// Mitsubishi GX Works2 project: SmartFarmDXnotST   PLC: FX3U/FX3UC

// global labels: Global1
VAR_GLOBAL
  AmbSens1_Humid AT D10 : INT;
  AmbSens1_Temp AT D11 : INT;
  AmbSens2_Humid AT D12 : INT;
  AmbSens2_Temp AT D13 : INT;
  SoilSens1_moist AT D20 : INT;
  SoilSens1_temp AT D21 : INT;
  SoilSens1_cond AT D22 : INT;
  SoilSens1_PH AT D23 : INT;
  SoilSens1_N AT D24 : INT;
  SoilSens1_P AT D25 : INT;
  SoilSens1_K AT D26 : INT;
  TempCon1_minT AT D30 : INT;
  TempCon1_maxT AT D31 : INT;
  TempCon1_Flg AT M10 : BOOL;
  TempCon1_Hs AT D32 : INT;
  TempCon1_Ms AT D33 : INT;
  TempCon1_Ss AT D34 : INT;
  TempCon1_He AT D35 : INT;
  TempCon1_Me AT D36 : INT;
  TempCon1_Se AT D37 : INT;
  TempCon2_minT AT D38 : INT;
  TempCon2_maxT AT D39 : INT;
  TempCon2_Flg AT M20 : BOOL;
  TempCon2_Hs AT D40 : INT;
  TempCon2_Ms AT D41 : INT;
  TempCon2_Ss AT D42 : INT;
  TempCon2_He AT D43 : INT;
  TempCon2_Me AT D44 : INT;
  TempCon2_Se AT D45 : INT;
  HumidCon1_minH AT D46 : INT;
  HumidCon1_maxH AT D47 : INT;
  HumidCon1_Flg AT M30 : BOOL;
  HumidCon1_Hs AT D48 : INT;
  HumidCon1_Ms AT D49 : INT;
  HumidCon1_Ss AT D50 : INT;
  HumidCon1_He AT D51 : INT;
  HumidCon1_Me AT D52 : INT;
  HumidCon1_Se AT D53 : INT;
  HumidCon2_minH AT D54 : INT;
  HumidCon2_maxH AT D55 : INT;
  HumidCon2_Flg AT M40 : BOOL;
  HumidCon2_Hs AT D56 : INT;
  HumidCon2_Ms AT D57 : INT;
  HumidCon2_Ss AT D58 : INT;
  HumidCon2_He AT D59 : INT;
  HumidCon2_Me AT D60 : INT;
  HumidCon2_Se AT D61 : INT;
  TimeCon1_Flg AT M50 : BOOL;
  TimeCon1_Hs AT D62 : INT;
  TimeCon1_Ms AT D63 : INT;
  TimeCon1_Ss AT D64 : INT;
  TimeCon1_He AT D65 : INT;
  TimeCon1_Me AT D66 : INT;
  TimeCon1_Se AT D67 : INT;
  TimeCon2_Flg AT M60 : BOOL;
  TimeCon2_Hs AT D68 : INT;
  TimeCon2_Ms AT D69 : INT;
  TimeCon2_Ss AT D70 : INT;
  TimeCon2_He AT D71 : INT;
  TimeCon2_Me AT D72 : INT;
  TimeCon2_Se AT D73 : INT;
  TimeCon3_Flg AT M70 : BOOL;
  TimeCon3_Hs AT D74 : INT;
  TimeCon3_Ms AT D75 : INT;
  TimeCon3_Ss AT D76 : INT;
  TimeCon3_He AT D77 : INT;
  TimeCon3_Me AT D78 : INT;
  TimeCon3_Se AT D79 : INT;
  TimeCon4_Flg AT M80 : BOOL;
  TimeCon4_Hs AT D80 : INT;
  TimeCon4_Ms AT D81 : INT;
  TimeCon4_Ss AT D82 : INT;
  TimeCon4_He AT D83 : INT;
  TimeCon4_Me AT D84 : INT;
  TimeCon4_Se AT D85 : INT;
  v0_enb AT M100 : BOOL;
  v0_mode_slc AT M101 : BOOL;
  v0_man_OD AT M102 : BOOL;
  v0_Temp1 AT M103 : BOOL;
  v0_Temp2 AT M104 : BOOL;
  v0_Humid1 AT M105 : BOOL;
  v0_Humid2 AT M106 : BOOL;
  v0_Time1 AT M107 : BOOL;
  v0_Time2 AT M108 : BOOL;
  v0_Time3 AT M109 : BOOL;
  v0_Time4 AT M110 : BOOL;
  v0_AMB_config AT M111 : BOOL;
  v0_TIME_config AT M112 : BOOL;
  v0_con_kill_flg AT M113 : BOOL;
  v0_con_pass_flg AT M114 : BOOL;
  v0_Drv_flg AT M115 : BOOL;
  v0_Yman_OD AT M116 : BOOL;
  v0_run_dur AT D100 : INT;
  v0_rest_dur AT D101 : INT;
  v1_enb AT M130 : BOOL;
  v1_mode_slc AT M131 : BOOL;
  v1_man_OD AT M132 : BOOL;
  v1_Temp1 AT M133 : BOOL;
  v1_Temp2 AT M134 : BOOL;
  v1_Humid1 AT M135 : BOOL;
  v1_Humid2 AT M136 : BOOL;
  v1_Time1 AT M137 : BOOL;
  v1_Time2 AT M138 : BOOL;
  v1_Time3 AT M139 : BOOL;
  v1_Time4 AT M140 : BOOL;
  v1_AMB_config AT M141 : BOOL;
  v1_TIME_config AT M142 : BOOL;
  v1_con_kill_flg AT M143 : BOOL;
  v1_con_pass_flg AT M144 : BOOL;
  v1_Drv_flg AT M145 : BOOL;
  v1_Yman_OD AT M146 : BOOL;
  v1_run_dur AT D102 : INT;
  v1_rest_dur AT D103 : INT;
END_VAR

PROGRAM MAIN
VAR
  AmbientSenseRea1 : AmbientSenseRead;
  SoilSenseRead_1 : SoilSenseRead;
  TempCon_1 : TempCon;
  TempCon_2 : TempCon;
  HumidCon_1 : HumidCon;
  HumidCon_2 : HumidCon;
  TimeCon_1 : TimeCon;
  TimeCon_2 : TimeCon;
  TimeCon_3 : TimeCon;
  TimeCon_4 : TimeCon;
  Valve_1 : Valve;
END_VAR
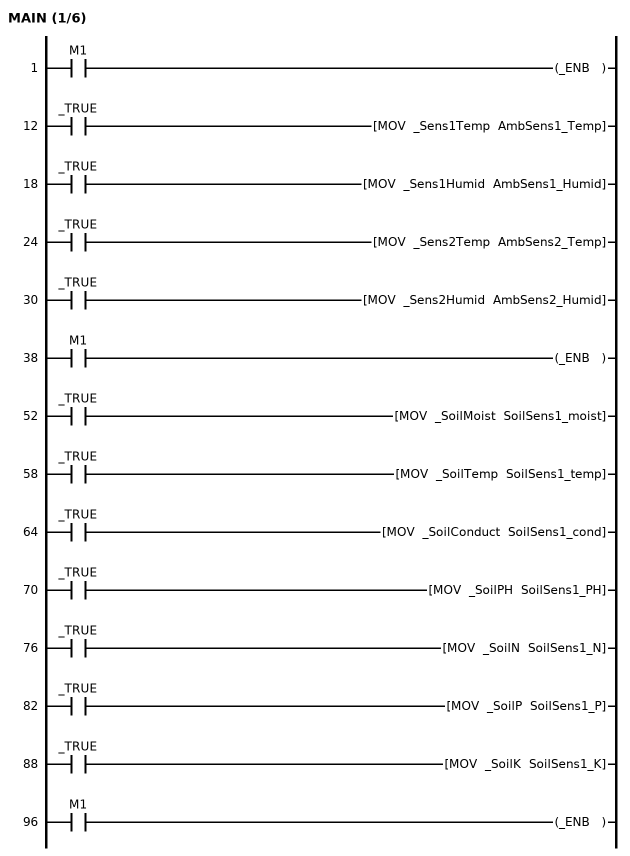
; FB BLK START AmbientSenseRead(AmbientSenseRea1)
1     LD      M1
      OUT     _ENB
; FB START
; FB_NAME AmbientSenseRead
; INSTANCE_NAME AmbientSenseRea1
; FB IN_B:ENB
; FB OUT_Sens1Temp:W
; FB OUT_Sens1Humid:W
; FB OUT_Sens2Temp:W
; FB OUT_Sens2Humid:W
; FB END
12    LD      _TRUE
      MOV     _Sens1Temp AmbSens1_Temp
18    LD      _TRUE
      MOV     _Sens1Humid AmbSens1_Humid
24    LD      _TRUE
      MOV     _Sens2Temp AmbSens2_Temp
30    LD      _TRUE
      MOV     _Sens2Humid AmbSens2_Humid
; FB BLK END
; FB BLK START SoilSenseRead(SoilSenseRead_1)
38    LD      M1
      OUT     _ENB
; FB START
; FB_NAME SoilSenseRead
; INSTANCE_NAME SoilSenseRead_1
; FB IN_B:ENB
; FB OUT_SoilMoist:W
; FB OUT_SoilTemp:W
; FB OUT_SoilConduct:W
; FB OUT_SoilPH:W
; FB OUT_SoilN:W
; FB OUT_SoilP:W
; FB OUT_SoilK:W
; FB END
52    LD      _TRUE
      MOV     _SoilMoist SoilSens1_moist
58    LD      _TRUE
      MOV     _SoilTemp SoilSens1_temp
64    LD      _TRUE
      MOV     _SoilConduct SoilSens1_cond
70    LD      _TRUE
      MOV     _SoilPH SoilSens1_PH
76    LD      _TRUE
      MOV     _SoilN SoilSens1_N
82    LD      _TRUE
      MOV     _SoilP SoilSens1_P
88    LD      _TRUE
      MOV     _SoilK SoilSens1_K
; FB BLK END
; FB BLK START TempCon(TempCon_1)
96    LD      M1
      OUT     _ENB
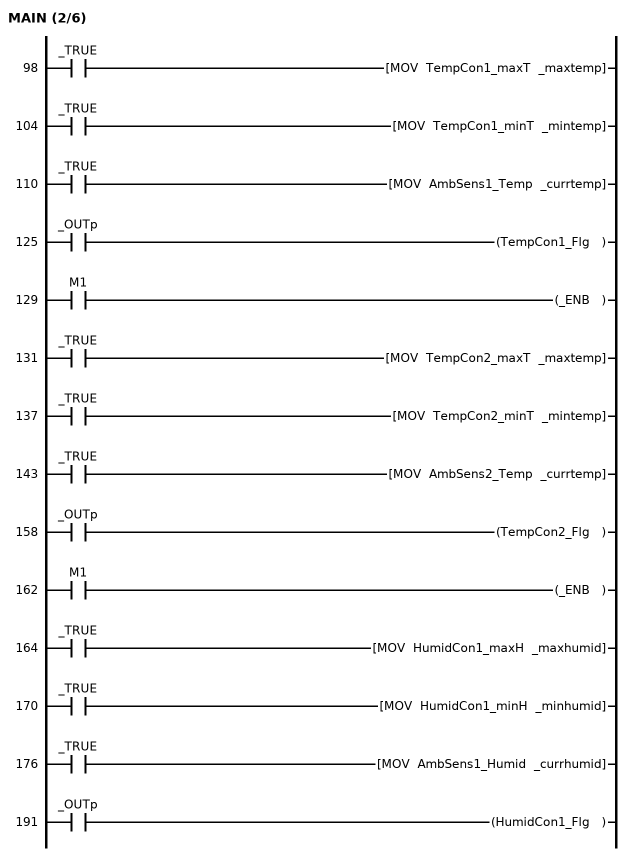
98    LD      _TRUE
      MOV     TempCon1_maxT _maxtemp
104   LD      _TRUE
      MOV     TempCon1_minT _mintemp
110   LD      _TRUE
      MOV     AmbSens1_Temp _currtemp
; FB START
; FB_NAME TempCon
; INSTANCE_NAME TempCon_1
; FB IN_B:ENB
; FB OUT_OUTp:B
; FB IN_W:maxtemp
; FB IN_W:mintemp
; FB IN_W:currtemp
; FB END
125   LD      _OUTp
      OUT     TempCon1_Flg
; FB BLK END
; FB BLK START TempCon(TempCon_2)
129   LD      M1
      OUT     _ENB
131   LD      _TRUE
      MOV     TempCon2_maxT _maxtemp
137   LD      _TRUE
      MOV     TempCon2_minT _mintemp
143   LD      _TRUE
      MOV     AmbSens2_Temp _currtemp
; FB START
; FB_NAME TempCon
; INSTANCE_NAME TempCon_2
; FB IN_B:ENB
; FB OUT_OUTp:B
; FB IN_W:maxtemp
; FB IN_W:mintemp
; FB IN_W:currtemp
; FB END
158   LD      _OUTp
      OUT     TempCon2_Flg
; FB BLK END
; FB BLK START HumidCon(HumidCon_1)
162   LD      M1
      OUT     _ENB
164   LD      _TRUE
      MOV     HumidCon1_maxH _maxhumid
170   LD      _TRUE
      MOV     HumidCon1_minH _minhumid
176   LD      _TRUE
      MOV     AmbSens1_Humid _currhumid
; FB START
; FB_NAME HumidCon
; INSTANCE_NAME HumidCon_1
; FB IN_B:ENB
; FB OUT_OUTp:B
; FB IN_W:maxhumid
; FB IN_W:minhumid
; FB IN_W:currhumid
; FB END
191   LD      _OUTp
      OUT     HumidCon1_Flg
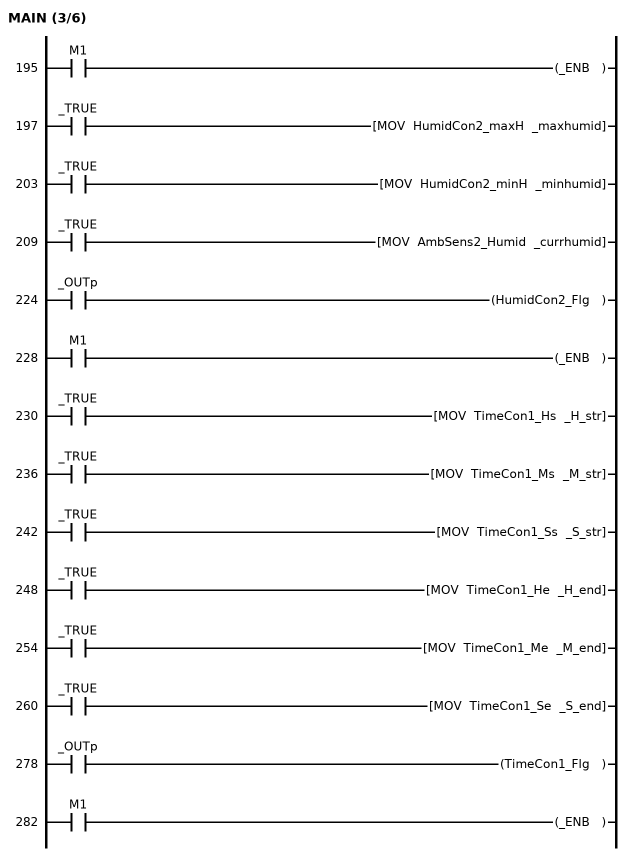
; FB BLK END
; FB BLK START HumidCon(HumidCon_2)
195   LD      M1
      OUT     _ENB
197   LD      _TRUE
      MOV     HumidCon2_maxH _maxhumid
203   LD      _TRUE
      MOV     HumidCon2_minH _minhumid
209   LD      _TRUE
      MOV     AmbSens2_Humid _currhumid
; FB START
; FB_NAME HumidCon
; INSTANCE_NAME HumidCon_2
; FB IN_B:ENB
; FB OUT_OUTp:B
; FB IN_W:maxhumid
; FB IN_W:minhumid
; FB IN_W:currhumid
; FB END
224   LD      _OUTp
      OUT     HumidCon2_Flg
; FB BLK END
; FB BLK START TimeCon(TimeCon_1)
228   LD      M1
      OUT     _ENB
230   LD      _TRUE
      MOV     TimeCon1_Hs _H_str
236   LD      _TRUE
      MOV     TimeCon1_Ms _M_str
242   LD      _TRUE
      MOV     TimeCon1_Ss _S_str
248   LD      _TRUE
      MOV     TimeCon1_He _H_end
254   LD      _TRUE
      MOV     TimeCon1_Me _M_end
260   LD      _TRUE
      MOV     TimeCon1_Se _S_end
; FB START
; FB_NAME TimeCon
; INSTANCE_NAME TimeCon_1
; FB IN_B:ENB
; FB OUT_OUTp:B
; FB IN_W:H_str
; FB IN_W:M_str
; FB IN_W:S_str
; FB IN_W:H_end
; FB IN_W:M_end
; FB IN_W:S_end
; FB END
278   LD      _OUTp
      OUT     TimeCon1_Flg
; FB BLK END
; FB BLK START TimeCon(TimeCon_2)
282   LD      M1
      OUT     _ENB
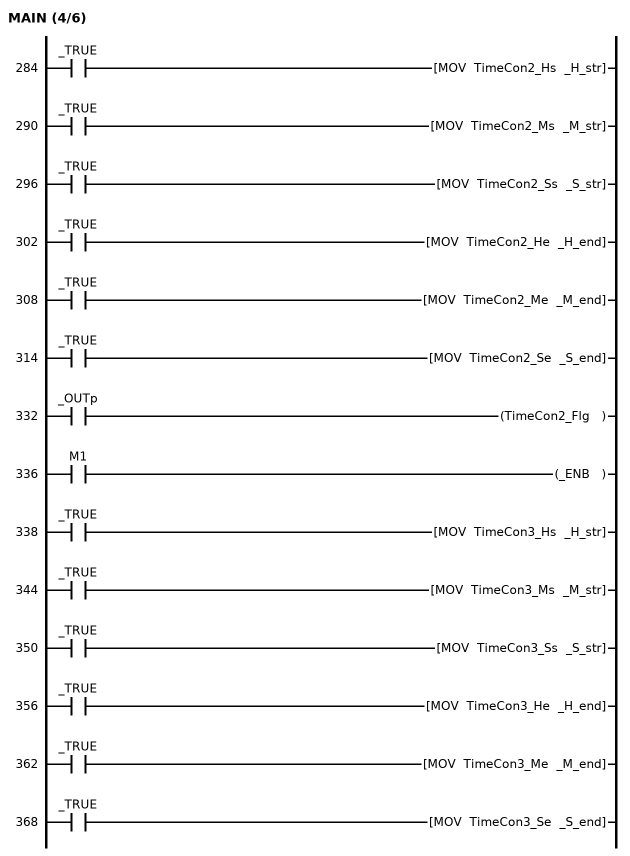
284   LD      _TRUE
      MOV     TimeCon2_Hs _H_str
290   LD      _TRUE
      MOV     TimeCon2_Ms _M_str
296   LD      _TRUE
      MOV     TimeCon2_Ss _S_str
302   LD      _TRUE
      MOV     TimeCon2_He _H_end
308   LD      _TRUE
      MOV     TimeCon2_Me _M_end
314   LD      _TRUE
      MOV     TimeCon2_Se _S_end
; FB START
; FB_NAME TimeCon
; INSTANCE_NAME TimeCon_2
; FB IN_B:ENB
; FB OUT_OUTp:B
; FB IN_W:H_str
; FB IN_W:M_str
; FB IN_W:S_str
; FB IN_W:H_end
; FB IN_W:M_end
; FB IN_W:S_end
; FB END
332   LD      _OUTp
      OUT     TimeCon2_Flg
; FB BLK END
; FB BLK START TimeCon(TimeCon_3)
336   LD      M1
      OUT     _ENB
338   LD      _TRUE
      MOV     TimeCon3_Hs _H_str
344   LD      _TRUE
      MOV     TimeCon3_Ms _M_str
350   LD      _TRUE
      MOV     TimeCon3_Ss _S_str
356   LD      _TRUE
      MOV     TimeCon3_He _H_end
362   LD      _TRUE
      MOV     TimeCon3_Me _M_end
368   LD      _TRUE
      MOV     TimeCon3_Se _S_end
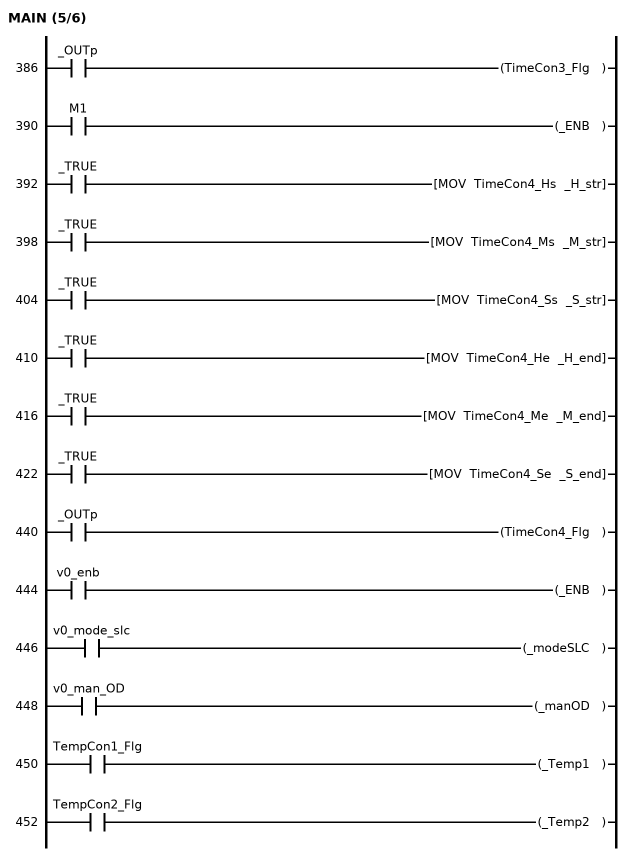
; FB START
; FB_NAME TimeCon
; INSTANCE_NAME TimeCon_3
; FB IN_B:ENB
; FB OUT_OUTp:B
; FB IN_W:H_str
; FB IN_W:M_str
; FB IN_W:S_str
; FB IN_W:H_end
; FB IN_W:M_end
; FB IN_W:S_end
; FB END
386   LD      _OUTp
      OUT     TimeCon3_Flg
; FB BLK END
; FB BLK START TimeCon(TimeCon_4)
390   LD      M1
      OUT     _ENB
392   LD      _TRUE
      MOV     TimeCon4_Hs _H_str
398   LD      _TRUE
      MOV     TimeCon4_Ms _M_str
404   LD      _TRUE
      MOV     TimeCon4_Ss _S_str
410   LD      _TRUE
      MOV     TimeCon4_He _H_end
416   LD      _TRUE
      MOV     TimeCon4_Me _M_end
422   LD      _TRUE
      MOV     TimeCon4_Se _S_end
; FB START
; FB_NAME TimeCon
; INSTANCE_NAME TimeCon_4
; FB IN_B:ENB
; FB OUT_OUTp:B
; FB IN_W:H_str
; FB IN_W:M_str
; FB IN_W:S_str
; FB IN_W:H_end
; FB IN_W:M_end
; FB IN_W:S_end
; FB END
440   LD      _OUTp
      OUT     TimeCon4_Flg
; FB BLK END
; FB BLK START Valve(Valve_1)
444   LD      v0_enb
      OUT     _ENB
446   LD      v0_mode_slc
      OUT     _modeSLC
448   LD      v0_man_OD
      OUT     _manOD
450   LD      TempCon1_Flg
      OUT     _Temp1
452   LD      TempCon2_Flg
      OUT     _Temp2
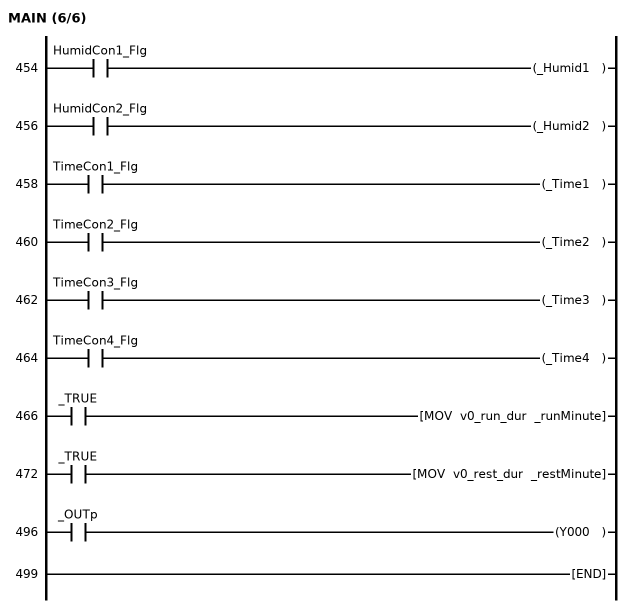
454   LD      HumidCon1_Flg
      OUT     _Humid1
456   LD      HumidCon2_Flg
      OUT     _Humid2
458   LD      TimeCon1_Flg
      OUT     _Time1
460   LD      TimeCon2_Flg
      OUT     _Time2
462   LD      TimeCon3_Flg
      OUT     _Time3
464   LD      TimeCon4_Flg
      OUT     _Time4
466   LD      _TRUE
      MOV     v0_run_dur _runMinute
472   LD      _TRUE
      MOV     v0_rest_dur _restMinute
; FB START
; FB_NAME Valve
; INSTANCE_NAME Valve_1
; FB IN_B:ENB
; FB OUT_OUTp:B
; FB IN_B:modeSLC
; FB IN_B:manOD
; FB IN_B:Temp1
; FB IN_B:Temp2
; FB IN_B:Humid1
; FB IN_B:Humid2
; FB IN_B:Time1
; FB IN_B:Time2
; FB IN_B:Time3
; FB IN_B:Time4
; FB IN_W:runMinute
; FB IN_W:restMinute
; FB END
496   LD      _OUTp
      OUT     Y000
; FB BLK END
499   END
END_PROGRAM

FUNCTION_BLOCK TimeCon
VAR_INPUT
  ENB : BOOL;
END_VAR
VAR_OUTPUT
  OUTp : BOOL;
END_VAR
VAR_INPUT
  H_str : INT;
  M_str : INT;
  S_str : INT;
  H_end : INT;
  M_end : INT;
  S_end : INT;
END_VAR
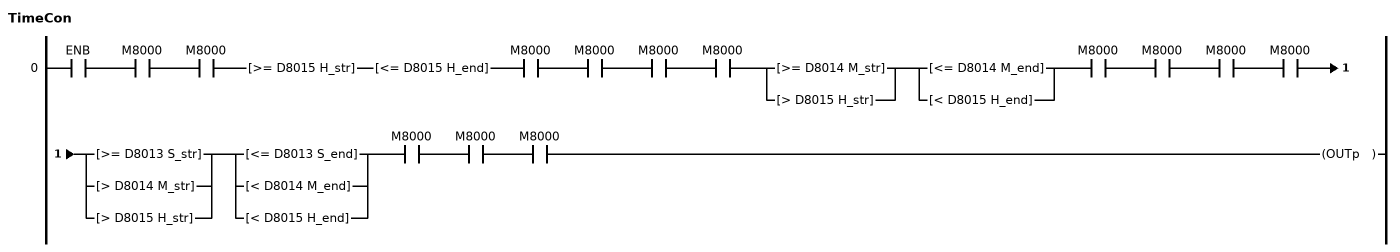
0     LD      ENB
      AND     M8000
      AND     M8000
      AND>=   D8015 H_str
      AND<=   D8015 H_end
      AND     M8000
      AND     M8000
      AND     M8000
      AND     M8000
      LD>=    D8014 M_str
      OR>     D8015 H_str
      ANB
      LD<=    D8014 M_end
      OR<     D8015 H_end
      ANB
      AND     M8000
      AND     M8000
      AND     M8000
      AND     M8000
      LD>=    D8013 S_str
      OR>     D8014 M_str
      OR>     D8015 H_str
      ANB
      LD<=    D8013 S_end
      OR<     D8014 M_end
      OR<     D8015 H_end
      ANB
      AND     M8000
      AND     M8000
      AND     M8000
      OUT     OUTp
END_FUNCTION_BLOCK

FUNCTION_BLOCK TempCon
VAR_INPUT
  ENB : BOOL;
END_VAR
VAR_OUTPUT
  OUTp : BOOL;
END_VAR
VAR_INPUT
  maxtemp : INT;
  mintemp : INT;
  currtemp : INT;
END_VAR
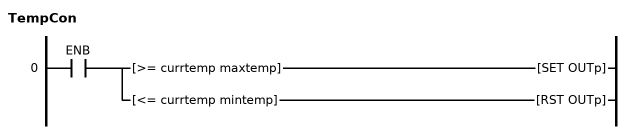
0     LD      ENB
      MPS
      AND>=   currtemp maxtemp
      SET     OUTp
      MPP
      AND<=   currtemp mintemp
      RST     OUTp
END_FUNCTION_BLOCK

FUNCTION_BLOCK HumidCon
VAR_INPUT
  ENB : BOOL;
  maxhumid : INT;
  minhumid : INT;
  currhumid : INT;
END_VAR
VAR_OUTPUT
  OUTp : BOOL;
END_VAR
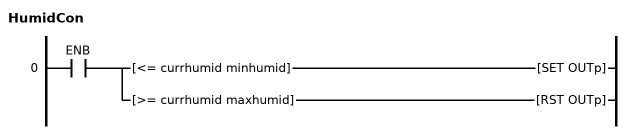
0     LD      ENB
      MPS
      AND<=   currhumid minhumid
      SET     OUTp
      MPP
      AND>=   currhumid maxhumid
      RST     OUTp
END_FUNCTION_BLOCK

FUNCTION_BLOCK AmbientSenseRead
VAR_INPUT
  ENB : BOOL;
END_VAR
VAR_OUTPUT
  Sens1Temp : INT;
  Sens1Humid : INT;
  Sens2Temp : INT;
  Sens2Humid : INT;
END_VAR
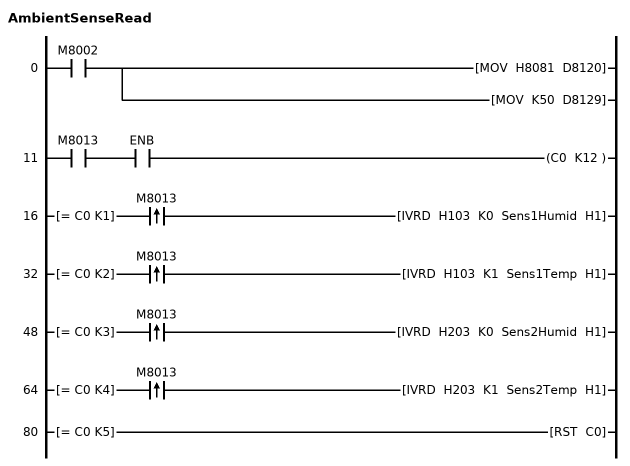
0     LD      M8002
      MOV     H8081 D8120
      MOV     K50 D8129
11    LD      M8013
      AND     ENB
      OUT     C0 K12
16    LD=     C0 K1
      ANDP    M8013
      IVRD    H103 K0 Sens1Humid H1
32    LD=     C0 K2
      ANDP    M8013
      IVRD    H103 K1 Sens1Temp H1
48    LD=     C0 K3
      ANDP    M8013
      IVRD    H203 K0 Sens2Humid H1
64    LD=     C0 K4
      ANDP    M8013
      IVRD    H203 K1 Sens2Temp H1
80    LD=     C0 K5
      RST     C0
END_FUNCTION_BLOCK

FUNCTION_BLOCK SoilSenseRead
VAR_INPUT
  ENB : BOOL;
END_VAR
VAR_OUTPUT
  SoilMoist : INT;
  SoilTemp : INT;
  SoilConduct : INT;
  SoilPH : INT;
  SoilN : INT;
  SoilP : INT;
  SoilK : INT;
END_VAR
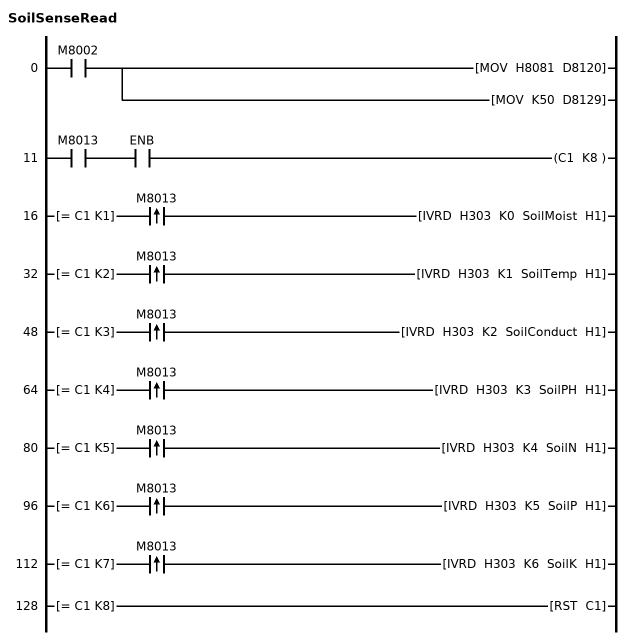
0     LD      M8002
      MOV     H8081 D8120
      MOV     K50 D8129
11    LD      M8013
      AND     ENB
      OUT     C1 K8
16    LD=     C1 K1
      ANDP    M8013
      IVRD    H303 K0 SoilMoist H1
32    LD=     C1 K2
      ANDP    M8013
      IVRD    H303 K1 SoilTemp H1
48    LD=     C1 K3
      ANDP    M8013
      IVRD    H303 K2 SoilConduct H1
64    LD=     C1 K4
      ANDP    M8013
      IVRD    H303 K3 SoilPH H1
80    LD=     C1 K5
      ANDP    M8013
      IVRD    H303 K4 SoilN H1
96    LD=     C1 K6
      ANDP    M8013
      IVRD    H303 K5 SoilP H1
112   LD=     C1 K7
      ANDP    M8013
      IVRD    H303 K6 SoilK H1
128   LD=     C1 K8
      RST     C1
END_FUNCTION_BLOCK

FUNCTION_BLOCK Valve
VAR_INPUT
  ENB : BOOL;
  modeSLC : BOOL;
  manOD : BOOL;
  Temp1 : BOOL;
  Temp2 : BOOL;
  Humid1 : BOOL;
  Humid2 : BOOL;
  Time1 : BOOL;
  Time3 : BOOL;
  Time2 : BOOL;
  Time4 : BOOL;
END_VAR
VAR_OUTPUT
  OUTp : BOOL;
END_VAR
VAR
  valveRunOD : BOOL;
  valveResting : BOOL;
  passCon : BOOL;
END_VAR
VAR_INPUT
  runMinute : INT;
END_VAR
VAR
  valveRunning : BOOL;
END_VAR
VAR_INPUT
  restMinute : INT;
END_VAR
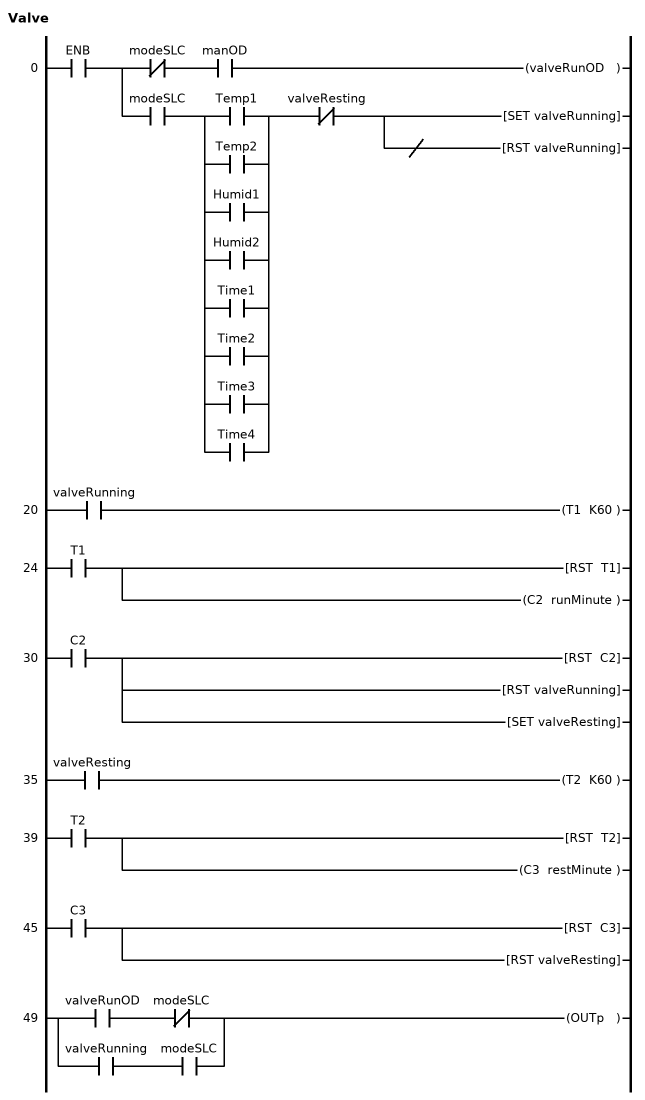
0     LD      ENB
      MPS
      ANI     modeSLC
      AND     manOD
      OUT     valveRunOD
      MPP
      AND     modeSLC
      LD      Temp1
      OR      Temp2
      OR      Humid1
      OR      Humid2
      OR      Time1
      OR      Time2
      OR      Time3
      OR      Time4
      ANB
      ANI     valveResting
      SET     valveRunning
      INV
      RST     valveRunning
20    LD      valveRunning
      OUT     T1 K60
24    LD      T1
      RST     T1
      OUT     C2 runMinute
30    LD      C2
      RST     C2
      RST     valveRunning
      SET     valveResting
35    LD      valveResting
      OUT     T2 K60
39    LD      T2
      RST     T2
      OUT     C3 restMinute
45    LD      C3
      RST     C3
      RST     valveResting
49    LD      valveRunOD
      ANI     modeSLC
      LD      valveRunning
      AND     modeSLC
      ORB
      OUT     OUTp
END_FUNCTION_BLOCK
